(* CODESYS project Frakta BSK Bus-Modul.export

Project tree, tasks and I/O mapping:
  Frakta/
    data type typFireDamperValues
    program FraktaMaster1 [ST]: onErrorCommunication
*)

// Frakta/typFireDamperValues
TYPE typFireDamperValues :
STRUCT
	// Bus Modul / Klappen (wichtigste Parameter)
	xDamper1Relay 							: BOOL;				// Status Relais Klappe 1 (0=Freigabe bzw. AUF / 1=ZU)
	xDamper2Relay 							: BOOL;				// Status Relais Klappe 2 (0=Freigabe bzw. AUF / 1=ZU)
	xDamper1OverrideEffective				: BOOL;				// Was auch immer Klappe 1...
	xDamper2OverrideEffective				: BOOL;				// Was auch immer Klappe 2...
	xDamper1Moving	 						: BOOL;				// Klappe 1 läuft
	xDamper2Moving	 						: BOOL;				// Klappe 2 läuft
	xDamper1Close	 						: BOOL;				// Klappe 1 Endschalter ZU
	xDamper1Open	 						: BOOL;				// Klappe 1 Endschalter AUF
	xDamper2Close	 						: BOOL;				// Klappe 2 Endschalter ZU
	xDamper2Open	 						: BOOL;				// Klappe 2 Endschalter AUF
	xDamper1FullAutoTest	 				: BOOL;				// Klappe 1 Testlauf durchführen, nur zurücklesen! (Statusmeldung bleibt bis Rücknahme anstehen)
	xDamper2FullAutoTest	 				: BOOL;				// Klappe 2 Testlauf durchführen, nur zurücklesen! (Statusmeldung bleibt bis Rücknahme anstehen)
	rDamper1CheckTime 						: REAL;				// Klappe 1 max. Laufzeit
	rDamper2CheckTime 						: REAL;				// Klappe 2 max. Laufzeit
	rDamper1SystemStatus					: REAL;				// Klappe 1 Status Meldung (0=Normal, 1=Endposition nicht erreicht, 5=sonstiges, 6=Testlauf aktiv, 7=Testlauf Normal, 8=Testlauf Fehler)
	rDamper2SystemStatus					: REAL;				// Klappe 2 Status Meldung (0=Normal, 1=Endposition nicht erreicht, 5=sonstiges, 6=Testlauf aktiv, 7=Testlauf Normal, 8=Testlauf Fehler)
	// Bus Modul selbst
	wSoftwareVersion 						: WORD;				// Software Version
	xFactoryDefault 						: BOOL;				// Werkseinstellungen Bus-Modul, nur zurücklesen!
	xClearMessage 							: BOOL;				// Was auch immer..., nur zurücklesen!
	rDelayAlarmCommunication				: REAL;				// Überwachungszeit Bus Kommunikation, nur zurücklesen! (30-120 sek., wenn die Kommunikation ausfällt, fahren die Klappen automatisch zu)
	xLogicAlarmCommunication 				: BOOL;				// Immer FALSE, gehört zur Bus Kommunikation (WatchDog)
	// Schreib Befehle	
	xSetLogicAlarmCommunication 			: BOOL := TRUE; 	// Dieser Wert muss immer geschrieben werden (WatchDog)
	xSetDamper1Relay 						: BOOL := FALSE;	// Vorgabe Relais Klappe 1 (0=Freigabe bzw. AUF / 1=ZU)	
	xSetDamper2Relay 						: BOOL := FALSE;	// Vorgabe Relais Klappe 2 (0=Freigabe bzw. AUF / 1=ZU)	
	xSetDamper1FullAutoTest	 				: BOOL := FALSE;	// Vorgabe Klappe 1 Testlauf durchführen (Statusmeldung bleibt bis Rücknahme anstehen)
	xSetDamper2FullAutoTest	 				: BOOL := FALSE;	// Vorgabe Klappe 2 Testlauf durchführen (Statusmeldung bleibt bis Rücknahme anstehen)
	xSetFactoryDefault 						: BOOL := FALSE;	// Vorgabe erkseinstellungen Bus-Modul
	xSetClearMessage 						: BOOL := FALSE;	// Was auch immer...
	rSetDamper1CheckTime					: REAL := 120;		// Vorgabe Klappe 1 max. Laufzeit
	rSetDamper2CheckTime					: REAL := 120;		// Vorgabe Klappe 2 max. Laufzeit
	rSetDelayAlarmCommunication				: REAL := 30;		// Vorgabe Überwachungszeit Bus Kommunikation, nur zurücklesen! (30-120 sek., wenn die Kommunikation ausfällt, fahren die Klappen automatisch zu)

	// RS485 Klemme / Wago
	xRS485ErrorCommunication				: BOOL;				// Fehler RS485 Kommunikation
	uiRS485ErrorCounter						: UINT;				// Fehler Zähler RS485 Kommunikation
	sRS485ErrorDescription					: STRING;			// Fehler Meldung RS485 Kommunikation
	
	// INTERN, Zwischenspeicher Wertänderung. 
	_xSetDamper1RelayOldValue 				: BOOL := TRUE;		// INTERN
	_xSetDamper2RelayOldValue 				: BOOL := TRUE;		// INTERN
	_xSetDamper1FullAutoTestOldValue	 	: BOOL := FALSE;	// INTERN
	_xSetDamper2FullAutoTestOldValue		: BOOL := FALSE;	// INTERN
	_xSetFactoryDefaultOldValue 			: BOOL := TRUE;		// INTERN
	_xSetClearMessageOldValue 				: BOOL := TRUE;		// INTERN
	_rSetDamper1CheckTimeOldValue			: REAL := 90;		// INTERN
	_rSetDamper2CheckTimeOldValue			: REAL := 90;		// INTERN
	_rSetDelayAlarmCommunicationOldValue	: REAL := 31;		// INTERN
END_STRUCT
END_TYPE

// Frakta/FraktaMaster1
PROGRAM FraktaMaster1 // Programm Frakta BSK Module auslesen maximal 32 Module je Master
VAR	
	// Einstellungen									
	SerialMaster  					: 	FbMbMasterSerial := (
							 			xConnect    := TRUE,
                                        udiBaudrate := 9600,
                                        usiDataBits := 8,
                                        eParity     := WagoTypesCom.eTTYParity.None,
                                        eStopBits   := WagoTypesCom.eTTYStopBits.One,
                                        eHandshake  := WagoTypesCom.eTTYHandshake.None,
                                        ePhysical   := WagoTypesCom.eTTYPhysicalLayer.RS485_HalfDuplex,
                                        eFrameType  := eMbFrameType.RTU,
                                        tTimeOut    := T#200MS
                                         );
	// Joblist Arraygröße = Anzahl der Module (max. 32), Init-Werte entsprechen den Modul-Adressen ... 
	bUnitIdModul					: 	ARRAY [1..2] OF BYTE := 
										[1,2];
	//Grenzwert Fehlerzähler bis xError TRUE wird	
	uiMaxErrorCounter				: 	UINT := 30;											 

	//Pause(-nzeit) zwischen den Abfragen und Schreib-Befehlen
	FbTonDelay        				: 	TON :=  (PT := T#50MS); 

	//sonstiges (ab hier muss nicht mehr eingestellt werden!)
	iJobNumber						: 	UINT := 1;								//aktueller Job											 
										 
	utQuery    						: 	typMbQuery := ( 
										bUnitId         := 0,       			// Adresse
                                   		bFunctionCode   := 3,   				// Funktion
                                   		uiReadAddress   := 0,       			// Startadresse
                                   		uiReadQuantity  := 42,      			// Anzahl
                                   		uiWriteAddress  := 0,       			// Startadresse
                                   		uiWriteQuantity := 0,       			// Anzahl
                                   		awWriteData     := [124(0)] 			// Schreib-Array
                                    	);
	utResponse      				: 	typMbResponse; 							// Anwort Telegramm RS485				
	xTxTrigger     					: 	BOOL;									// Ausführung starten RS485
  	xIsConnected					: 	BOOL;									// Verbunden RS485
		
	utModule						: 	ARRAY [1..32] OF typFireDamperValues;  	// Datenmodell Bus-Module, für max. 32 Bus-Module
										
	FbJobFinish						: 	F_TRIG;	 								// Flanke wenn Job beendet
	xWriteJob						:	BOOL 	:= FALSE; 						// Umschaltung zwischen lesen und schreiben 0=lesen / 1=schreiben 
	xJobFinish						: 	BOOL; 									// Job fertig
	xJobFinishRead 					: 	BOOL; 									// Lese Job fertig
	xJobsFinishWrite 				: 	BOOL; 									// Schreib Jobs fertig
	xChangeWriteValue				: 	ARRAY [1..32] OF BOOL;					// Wert-Änderung bei den Schreib-Befehlen
	iChangeWriteValue				: 	DINT;									// Schleife Rücksetzen xChangeWriteValue
	uiWriteAddress					:	UINT;
	arWriteAddress					: 	ARRAY [1..10] OF UINT := 				// Schreib Adressen Array,
										[42,7,8,25,26,27,28,34,35,41]; 			// Siehe Bus-Modul Beschreibung, Frakta
	iWriteJobNumber					: 	INT := 1;
	
END_VAR

//Debug Bereich Schreibbefehle testen
utModule[1].xSetDamper1Relay;
utModule[1].xSetDamper2Relay;
utModule[1].xSetDamper1FullAutoTest;
utModule[1].xSetDamper2FullAutoTest;
utModule[1].xSetFactoryDefault;
utModule[1].xSetClearMessage;
utModule[1].rSetDamper1CheckTime;
utModule[1].rSetDamper2CheckTime;
utModule[1].rSetDelayAlarmCommunication;


//Limits überwachen ("upper_bound", Größe vom Array bestimmen)
IF  iJobNumber<1 OR iJobNumber > UPPER_BOUND(bUnitIdModul,1) THEN
	iJobNumber:=1;
END_IF
IF  iWriteJobNumber<1 OR iWriteJobNumber > UPPER_BOUND(arWriteAddress,1) THEN
	iWriteJobNumber:=1;
END_IF
		

// richtige Moduladressen übergeben
utQuery.bUnitId:= bUnitIdModul[iJobNumber]; 

// Umschaltung zwischen lesen und schreiben
utQuery.bFunctionCode		:= SEL	(xWriteJob, 3, 6);
utQuery.uiReadAddress		:= SEL	(xWriteJob, 0, 0);
utQuery.uiReadQuantity		:= SEL	(xWriteJob, 42, 0);
utQuery.uiWriteAddress		:= SEL	(xWriteJob, 0, uiWriteAddress);
utQuery.uiWriteQuantity		:= SEL	(xWriteJob, 0, 1);

// Funktionsblock Seriale Schnittstelle aufrufen
SerialMaster(
	I_Port:= 		COM2, 
	xIsConnected=> 	xIsConnected, 
	utQuery:= 		utQuery, 
	xTrigger:= 		xTxTrigger, 
	utResponse:= 	utResponse
);


// wenn verbunden dann abfragen, kurze Pause zwischen den Abfragen
IF xIsConnected THEN
	FbTonDelay( 
		IN := (NOT FbTonDelay.Q) AND (NOT xTxTrigger)
			);
	xTxTrigger S= FbTonDelay.Q; 

	FbJobFinish(
			CLK:= xTxTrigger, 
			Q=> xJobFinish
		);
	
	xJobFinishRead:= 				xJobFinish AND NOT xWriteJob;	
	xJobsFinishWrite:= 			xJobFinish AND  xWriteJob;
	
	IF xJobFinishRead THEN
				// Kommunikationsfehler eintragen bzw. rücksetzen
				utModule[iJobNumber].xRS485ErrorCommunication			:= utModule[iJobNumber].uiRS485ErrorCounter >= uiMaxErrorCounter; 	//Erst nach x Fehlern den Fehler melden	
				utModule[iJobNumber].sRS485ErrorDescription				:= SerialMaster.oStatus.sDescription; 							// Fehler Meldung aus der RS485 Kommunikation!
				IF utModule[iJobNumber].xRS485ErrorCommunication THEN	// Im Fehlerfall alle Werte zurücksetzen
					onErrorCommunication();							//Alle Variablen auf "null"
				END_IF
			IF NOT SerialMaster.xError THEN // Antwort Daten richtig eintragen
				utModule[iJobNumber].wSoftwareVersion				:= TO_WORD(utResponse.awData[0]);
				utModule[iJobNumber].xDamper1Relay 					:= TO_BOOL(utResponse.awData[7]);
				utModule[iJobNumber].xDamper2Relay 					:= TO_BOOL(utResponse.awData[8]);
				utModule[iJobNumber].xDamper1OverrideEffective 		:= TO_BOOL(utResponse.awData[15]);
				utModule[iJobNumber].xDamper2OverrideEffective 		:= TO_BOOL(utResponse.awData[16]);
				utModule[iJobNumber].xDamper1Moving	 				:= TO_BOOL(utResponse.awData[17]);
				utModule[iJobNumber].xDamper2Moving	 				:= TO_BOOL(utResponse.awData[18]);
				utModule[iJobNumber].xDamper1Close	 				:= TO_BOOL(utResponse.awData[21]);
				utModule[iJobNumber].xDamper1Open	 				:= TO_BOOL(utResponse.awData[22]);
				utModule[iJobNumber].xDamper2Close	 				:= TO_BOOL(utResponse.awData[23]);
				utModule[iJobNumber].xDamper2Open	 				:= TO_BOOL(utResponse.awData[24]);
				utModule[iJobNumber].xDamper1FullAutoTest			:= TO_BOOL(utResponse.awData[25]);
				utModule[iJobNumber].xDamper2FullAutoTest			:= TO_BOOL(utResponse.awData[26]);
				utModule[iJobNumber].xFactoryDefault				:= TO_BOOL(utResponse.awData[27]);
				utModule[iJobNumber].xClearMessage					:= TO_BOOL(utResponse.awData[28]);
				utModule[iJobNumber].rDamper1CheckTime 				:= TO_REAL(utResponse.awData[34]);
				utModule[iJobNumber].rDamper2CheckTime 				:= TO_REAL(utResponse.awData[35]);
				utModule[iJobNumber].rDamper1SystemStatus			:= TO_REAL(utResponse.awData[36]);
				utModule[iJobNumber].rDamper2SystemStatus		 	:= TO_REAL(utResponse.awData[37]);
				utModule[iJobNumber].rDelayAlarmCommunication		:= TO_REAL(utResponse.awData[41]);
				utModule[iJobNumber].xLogicAlarmCommunication		:= TO_BOOL(utResponse.awData[42]);
				utModule[iJobNumber].uiRS485ErrorCounter					:= 0; // wenn kein Fehler mehr ist, Counter zurücksetzen
			ELSE
				// Im Fehlerfall den Fehlerzähler um eins erhöhen
				utModule[iJobNumber].uiRS485ErrorCounter					:= utModule[iJobNumber].uiRS485ErrorCounter + 1;
			END_IF

		// Auf schreiben umschalten
		xWriteJob:= TRUE;
	END_IF	
	IF xWriteJob THEN
		uiWriteAddress:= arWriteAddress[iWriteJobNumber];
			CASE iWriteJobNumber OF		
				1: // 42 Logic Alarm Communication (Dieser Wert muss immer geschreiben werden, WatchDog!)
					utQuery.awWriteData[0]:= TO_WORD(utModule[iJobNumber].xSetLogicAlarmCommunication);				
				2: // 7 SetRelay Damper 1
					utQuery.awWriteData[0]:= TO_WORD(utModule[iJobNumber].xSetDamper1Relay);
				3: // 2 SetRelay Damper 2
					utQuery.awWriteData[0]:= TO_WORD(utModule[iJobNumber].xSetDamper2Relay);
				4: // 25 FullAutoTest Damper 1
					utQuery.awWriteData[0]:= TO_WORD(utModule[iJobNumber].xSetDamper1FullAutoTest);
				5: // 26 FullAutoTest Damper 2
					utQuery.awWriteData[0]:= TO_WORD(utModule[iJobNumber].xSetDamper2FullAutoTest);
				6: // 27 SetFactoryDefault 
					utQuery.awWriteData[0]:= TO_WORD(utModule[iJobNumber].xSetFactoryDefault);
				7: // 28 Clear Message 
					utQuery.awWriteData[0]:= TO_WORD(utModule[iJobNumber].xSetClearMessage);
				8: // 34 Check Time Damper 1
					utQuery.awWriteData[0]:= TO_WORD(utModule[iJobNumber].rSetDamper1CheckTime);
				9: // 35 Check Time Damper 2 
					utQuery.awWriteData[0]:= TO_WORD(utModule[iJobNumber].rSetDamper2CheckTime);
				10: // 41 Delay Alarm Communication 
					utQuery.awWriteData[0]:= TO_WORD(utModule[iJobNumber].rSetDelayAlarmCommunication);
			ELSE
				utQuery.awWriteData[0]:= 0 ; 
				xWriteJob:= FALSE;
			END_CASE;	
		IF xJobsFinishWrite THEN 
		// 		Optimierung Schreib Befehle
		// 		xSetDamper1Relay
		IF utModule[iJobNumber].xSetDamper1Relay <>	utModule[iJobNumber]._xSetDamper1RelayOldValue THEN 	
			utModule[iJobNumber]._xSetDamper1RelayOldValue:= utModule[iJobNumber].xSetDamper1Relay;
			xChangeWriteValue[iJobNumber]:= TRUE;
		END_IF	
		// 		xSetDamper2Relay
		IF utModule[iJobNumber].xSetDamper2Relay <>	utModule[iJobNumber]._xSetDamper2RelayOldValue THEN	
			utModule[iJobNumber]._xSetDamper2RelayOldValue:= utModule[iJobNumber].xSetDamper2Relay;
			xChangeWriteValue[iJobNumber]:= TRUE;
		END_IF
		//		xSetDamper1FullAutoTest
		IF utModule[iJobNumber].xSetDamper1FullAutoTest <>	utModule[iJobNumber]._xSetDamper1FullAutoTestOldValue THEN
			utModule[iJobNumber]._xSetDamper1FullAutoTestOldValue:= utModule[iJobNumber].xSetDamper1FullAutoTest;
			xChangeWriteValue[iJobNumber]:= TRUE;
		END_IF
		//		xSetDamper2FullAutoTest
		IF utModule[iJobNumber].xSetDamper2FullAutoTest <>	utModule[iJobNumber]._xSetDamper2FullAutoTestOldValue THEN
			utModule[iJobNumber]._xSetDamper2FullAutoTestOldValue:= utModule[iJobNumber].xSetDamper2FullAutoTest;
			xChangeWriteValue[iJobNumber]:= TRUE;
		END_IF
		//		xSetFactoryDefault
		IF utModule[iJobNumber].xSetFactoryDefault <>	utModule[iJobNumber]._xSetFactoryDefaultOldValue THEN
			utModule[iJobNumber]._xSetFactoryDefaultOldValue:= utModule[iJobNumber].xSetFactoryDefault;
			xChangeWriteValue[iJobNumber]:= TRUE;
		END_IF
		//		xSetClearMessage
		IF utModule[iJobNumber].xSetClearMessage <>	utModule[iJobNumber]._xSetClearMessageOldValue THEN
			utModule[iJobNumber]._xSetClearMessageOldValue:= utModule[iJobNumber].xSetClearMessage;
			xChangeWriteValue[iJobNumber]:= TRUE;
		END_IF
		// 		rSetDamper1CheckTime
		IF utModule[iJobNumber].rSetDamper1CheckTime <>	utModule[iJobNumber]._rSetDamper1CheckTimeOldValue THEN
			utModule[iJobNumber]._rSetDamper1CheckTimeOldValue:= utModule[iJobNumber].rSetDamper1CheckTime;
			xChangeWriteValue[iJobNumber]:= TRUE;
		END_IF
		// 		rSetDamper2CheckTime
		IF utModule[iJobNumber].rSetDamper2CheckTime <>	utModule[iJobNumber]._rSetDamper2CheckTimeOldValue THEN
			utModule[iJobNumber]._rSetDamper2CheckTimeOldValue:= utModule[iJobNumber].rSetDamper2CheckTime;
			xChangeWriteValue[iJobNumber]:= TRUE;
		END_IF
		//		rSetDelayAlarmCommunication	
		IF utModule[iJobNumber].rSetDelayAlarmCommunication <>	utModule[iJobNumber]._rSetDelayAlarmCommunicationOldValue THEN
			utModule[iJobNumber]._rSetDelayAlarmCommunicationOldValue:= utModule[iJobNumber].rSetDelayAlarmCommunication;
			xChangeWriteValue[iJobNumber]:= TRUE;
		END_IF	
		
		// 		Schreib Job Zähler
		IF xChangeWriteValue[iJobNumber] THEN;
			iWriteJobNumber:= iWriteJobNumber + 1;					// Schreib Job Zähler + 1 (gleiches Bus-Modul)
		ELSE
			iWriteJobNumber:= 99;									// Wenn keine Änderung, dann WirteJobs abbrechen (99)
		END_IF
		//	IF NOT onChangeWriteValue(xChangeAccepted) THEN			// Schreib Optimierung
		//		iWriteJobNumber:= 99;								// Wenn keine Änderung, dann WirteJobs abbrechen (99)
		//	END_IF
		END_IF
		IF xJobsFinishWrite AND iWriteJobNumber > UPPER_BOUND(arWriteAddress,1) THEN
			iJobNumber:= 		iJobNumber + 1;						// Job Zähler + 1
			xWriteJob:= 		FALSE;								// Schreib Job beenden
	
		// Optimierung
		FOR iChangeWriteValue:= 1 TO UPPER_BOUND(bUnitIdModul,1) BY 1 DO
			xChangeWriteValue[iChangeWriteValue]:= FALSE;		
		END_FOR
	
		//	xChangeAccepted:= TRUE;									//Alle Änderungen übernommen 
		END_IF
	END_IF
END_IF

METHOD onErrorCommunication // Im Fehlerfall alle gelesen Werte auf "0 / FALSE" setzen.
VAR_INPUT
END_VAR
utModule[iJobNumber].wSoftwareVersion				:= TO_WORD(0);
utModule[iJobNumber].xDamper1Relay 					:= TO_BOOL(0);
utModule[iJobNumber].xDamper2Relay 					:= TO_BOOL(0);
utModule[iJobNumber].xDamper1OverrideEffective 		:= TO_BOOL(0);
utModule[iJobNumber].xDamper2OverrideEffective 		:= TO_BOOL(0);
utModule[iJobNumber].xDamper1Moving	 				:= TO_BOOL(0);
utModule[iJobNumber].xDamper2Moving	 				:= TO_BOOL(0);
utModule[iJobNumber].xDamper1Close	 				:= TO_BOOL(0);
utModule[iJobNumber].xDamper1Open	 				:= TO_BOOL(0);
utModule[iJobNumber].xDamper2Close	 				:= TO_BOOL(0);
utModule[iJobNumber].xDamper2Open	 				:= TO_BOOL(0);
utModule[iJobNumber].rDamper1CheckTime 				:= TO_REAL(0);
utModule[iJobNumber].rDamper2CheckTime 				:= TO_REAL(0);
utModule[iJobNumber].rDamper1SystemStatus			:= TO_REAL(0);
utModule[iJobNumber].rDamper2SystemStatus		 	:= TO_REAL(0);
END_METHOD

END_PROGRAM
